TYPE ST_Control :
STRUCT
	ClearAllFaults : BOOL;
END_STRUCT
END_TYPE

(* stored: Version 1.1.0.1, ProductVersion 3.1.4024.11
   DUT ST_Control: Id {8c7fcd92-0695-4de1-b521-f46ddb30fe29} *)
